FUNCTION_BLOCK IA_VDS (* ISOBUS Adapter for Vehicle Direction/Speed (VDS) *)
  (* Standard: ISO 11783-7; Classification: PGN 65256; Description: Copyright (c) 2024-2026 HR Agrartechnik GmbH This program and the accompanying materials are made available under the terms of the Eclipse Public License 2.0 which is available at https://www.eclipse.org/legal/epl-2.0/ SPDX-License-Identifier: EPL-2.0 *)
  (* Version 1.0, 2026-04-19, Franz Höpfinger, HR Agrartechnik GmbH, initial API and implementation (Adapter Wrapper for I_VDS) *)
  PACKAGE isobus::tecu;
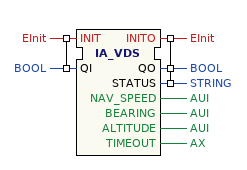
  EVENT_INPUT
    INIT : EInit WITH QI; (* Service Initialization *)
  END_EVENT
  EVENT_OUTPUT
    INITO : EInit WITH QO, STATUS; (* Initialization Confirm *)
  END_EVENT
  VAR_INPUT
    QI : BOOL; (* Event Input Qualifier *)
  END_VAR
  VAR_OUTPUT
    QO : BOOL; (* Event Output Qualifier *)
    STATUS : STRING;
  END_VAR
  PLUGS
    NAV_SPEED : adapter::types::unidirectional::AUI; (* Navigation-based vehicle speed *)
    BEARING : adapter::types::unidirectional::AUI; (* Compass bearing *)
    ALTITUDE : adapter::types::unidirectional::AUI; (* Altitude *)
    TIMEOUT : adapter::types::unidirectional::AX; (* Timeout Status *)
  END_PLUGS
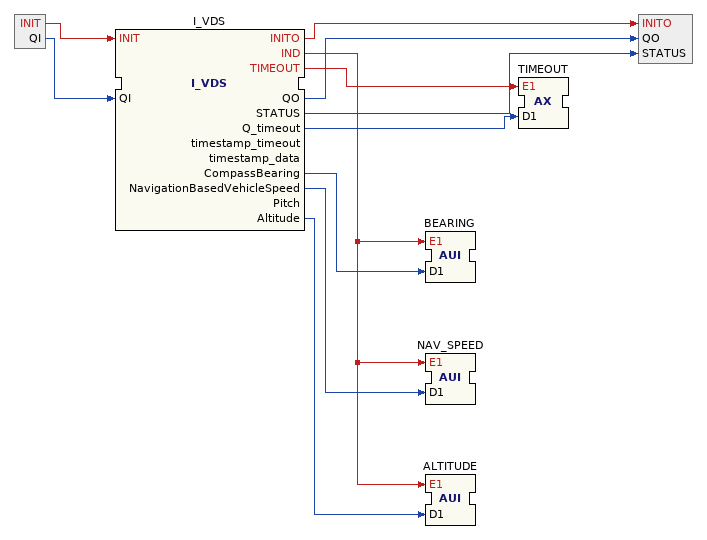
  FBS
    I_VDS : isobus::tecu::I_VDS;
  END_FBS
  EVENT_CONNECTIONS
    INIT TO I_VDS.INIT;
    I_VDS.INITO TO INITO;
    I_VDS.TIMEOUT TO TIMEOUT.E1;
    I_VDS.IND TO NAV_SPEED.E1;
    I_VDS.IND TO BEARING.E1;
    I_VDS.IND TO ALTITUDE.E1;
  END_CONNECTIONS
  DATA_CONNECTIONS
    QI TO I_VDS.QI;
    I_VDS.QO TO QO;
    I_VDS.STATUS TO STATUS;
    I_VDS.Q_timeout TO TIMEOUT.D1;
    I_VDS.NavigationBasedVehicleSpeed TO NAV_SPEED.D1;
    I_VDS.CompassBearing TO BEARING.D1;
    I_VDS.Altitude TO ALTITUDE.D1;
  END_CONNECTIONS
END_FUNCTION_BLOCK
